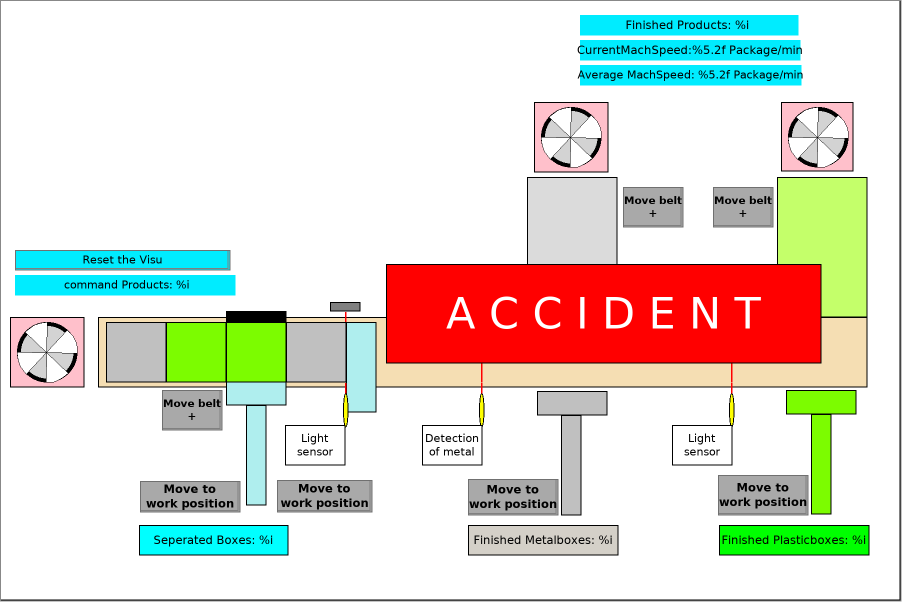
VISUALIZATION VIS_TemplateMachine  // 902x602
    Rectangle (0,0 900x600)
    Rectangle (98,317 769x70)
    Rectangle (777,177 90x140)
    Rectangle (527,177 90x140)
    Rectangle (716,302 30x9)
    Rectangle (467,302 30x9)
    Ellipse (479,393 5x34)
    Ellipse (729,393 5x34)
    Group (537,391 70x124)
        p2738717112: MAIN.fbVisu.fYMetal
        Rectangle (0,0 70x24)
        Rectangle (24,24 20x100)
    Group (787,391 70x124)
        p2738717112: MAIN.fbVisu.fYPlastic
        Rectangle (-1,-1 70x24)
        Rectangle (24,23 20x100)
    Group (227,382 60x124)
        p2738717112: MAIN.fbVisu.fYClamp
        Rectangle (19,23 20x100)
        Rectangle (-1,-1 60x24)
    Rectangle (106,322 60x60)
        p3560616238: MAIN.fbVisu.aBoxX[4]
        p2738717112: MAIN.fbVisu.aBoxY[4]
    Rectangle (226,322 60x60)
        p3560616238: MAIN.fbVisu.aBoxX[2]
        p2738717112: MAIN.fbVisu.aBoxY[2]
    Rectangle (166,322 60x60)
        p3560616238: MAIN.fbVisu.aBoxX[3]
        p2738717112: MAIN.fbVisu.aBoxY[3]
    Textfield (422,425 60x40), "Detection of metal"
    Textfield (672,425 60x40), "Light sensor"
    Rectangle (481,383 1x10)
    Rectangle (481,312 1x70)
    Rectangle (731,312 1x70)
    Rectangle (731,383 1x10)
    Button (623,187 60x40), "Move belt +", colour toggle: MAIN.fbVisu.bButtonColorMetalFw, invisible if: NOT (MAIN.fbMachine.eMode= 3), input disabled if: NOT (MAIN.fbMachine.eState = ePMLState_Execute)
        p573394764: MAIN.fbVisu.nButtonColorMetalFw
        toggle MAIN.fbVisu.bButtonMetalFwOut
    Button (713,187 60x40), "Move belt +", colour toggle: MAIN.fbVisu.bButtonColorPlasticFw, invisible if: NOT (MAIN.fbMachine.eMode= 3), input disabled if: NOT (MAIN.fbMachine.eState = ePMLState_Execute)
        p573394764: MAIN.fbVisu.nButtonColorPlasticFw
        toggle MAIN.fbVisu.bButtonPlasticFwOut
    Button (162,390 60x40), "Move belt +", colour toggle: MAIN.fbVisu.bButtonColorMainFw, invisible if: NOT (MAIN.fbMachine.eMode= 3), input disabled if: NOT (MAIN.fbMachine.eState = ePMLState_Execute)
        p573394764: MAIN.fbVisu.nButtonColorMainFw
        toggle MAIN.fbVisu.bButtonMainFwOut
    Button (277,480 95x32), "Move to work position", colour toggle: MAIN.fbVisu.bButtonColorBarrier, invisible if: NOT (MAIN.fbMachine.eMode= 3), input disabled if: NOT (MAIN.fbMachine.eState = ePMLState_Execute)
        p573394764: MAIN.fbVisu.nButtonColorBarrier
        toggle MAIN.fbVisu.bButtonBarrierToWorkOut
    Button (140,481 100x31), "Move to work position", colour toggle: MAIN.fbVisu.bButtonColorClamp, invisible if: NOT (MAIN.fbMachine.eMode= 3), input disabled if: NOT (MAIN.fbMachine.eState = ePMLState_Execute)
        p573394764: MAIN.fbVisu.nButtonColorClamp
        toggle MAIN.fbVisu.bButtonClampToWorkOut
    Button (468,479 90x36), "Move to work position", colour toggle: MAIN.fbVisu.bButtonColorMetalCyl, invisible if: NOT (MAIN.fbMachine.eMode= 3), input disabled if: NOT (MAIN.fbMachine.eState = ePMLState_Execute)
        p573394764: MAIN.fbVisu.nButtonColorMetalCyl
        toggle MAIN.fbVisu.bButtonMetalToWorkOut
    Button (718,475 90x40), "Move to work position", colour toggle: MAIN.fbVisu.bButtonColorPlasticCyl, invisible if: NOT (MAIN.fbMachine.eMode= 3), input disabled if: NOT (MAIN.fbMachine.eState = ePMLState_Execute)
        p573394764: MAIN.fbVisu.nButtonColorPlasticCyl
        toggle MAIN.fbVisu.bButtonPlasticToWorkOut
    Rectangle (346,322 30x90)
        p2738717112: MAIN.fbVisu.fYBarrier
    Rectangle (330,302 30x9)
    Ellipse (343,393 5x34)
    Rectangle (345,383 1x10)
    Rectangle (345,312 1x70)
    Textfield (285,425 60x40), "Light sensor"
    Rectangle (226,311 60x11)
    Rectangle (286,322 60x60)
        p3560616238: MAIN.fbVisu.aBoxX[1]
        p2738717112: MAIN.fbVisu.aBoxY[1]
    Rectangle (386,264 435x99), "A C C I D E N T", invisible if: NOT MAIN.fbVisu.bAccident
    Textfield (10,317 74x70)
    Rectangle (46,322 1x60)
    Rectangle (17,352 60x1)
    Ellipse (17,322 60x60)
    Polygon (47,322) (46,382) (53,382) (58,380) (63,377) (68,373) (25,332) (22,336) (20,340) (18,345) (17,352) (77,353) (77,347) (76,342) (73,336) (67,330) (26,374) (23,370) (20,366) (18,360) (17,353) (18,347) (19,342) (22,336) (26,331) (30,328) (34,325) (40,323)
        p2858320360: MAIN.fbVisu.nAngleMain
    Textfield (534,102 74x70)
    Rectangle (570,107 1x60)
    Rectangle (541,137 60x1)
    Ellipse (541,107 60x60)
    Polygon (571,107) (570,167) (577,167) (582,165) (587,162) (592,158) (549,117) (546,121) (544,125) (542,130) (541,137) (601,138) (601,132) (600,127) (597,121) (591,115) (550,159) (547,155) (544,151) (542,145) (541,138) (542,132) (543,127) (546,121) (550,116) (554,113) (558,110) (564,108)
        p2858320360: MAIN.fbVisu.nAngleMetal
    Textfield (781,102 72x69)
    Rectangle (817,107 1x60)
    Rectangle (788,137 60x1)
    Ellipse (788,107 60x60)
    Polygon (818,107) (817,167) (824,167) (829,165) (834,162) (839,158) (796,117) (793,121) (791,125) (789,130) (788,137) (848,138) (848,132) (847,127) (844,121) (838,115) (797,159) (794,155) (791,151) (789,145) (788,138) (789,132) (790,127) (793,121) (797,116) (801,113) (805,110) (811,108)
        p2858320360: MAIN.fbVisu.nAnglePlastic
    Rectangle (15,275 220x20), "command Products: %i", text variable: PackTags.Command.Parameter[2].Value, colour toggle: (MAIN.fbVisu.bInValidEntry OR PackTags.Admin.Warning[1].Trigger), invisible if: NOT ( MAIN.fbMachine.eMode = 1)
        OnMouseClick: write nVisuProductCommand via Default
    Rectangle (580,15 218x20), "Finished Products: %i", text variable: PackTags.Admin.ProdProcessedCount[1].Count, invisible if: NOT ( MAIN.fbMachine.eMode = 1)
    Button (15,250 215x20), "Reset the Visu", invisible if: (MAIN.fbMachine.eMode = 1 AND (MAIN.fbMachine.eState = ePMLState_Clearing OR MAIN.fbMachine.eState = ePMLState_Aborting OR MAIN.fbMachine.eState = ePMLState_Stopping OR MAIN.fbMachine.eState = ePMLState_Resetting OR MAIN.fbMachine.eState = ePMLState_Starting OR MAIN.fbMachine.eState = ePMLState_Execute OR MAIN.fbMachine.eState = ePMLState_Completing OR MAIN.fbMachine.eState = ePMLState_Suspending OR MAIN.fbMachine.eState = ePMLState_Holding))
        tap stChangeIntoProduction.bYesReset
    Rectangle (580,40 220x20), "CurrentMachSpeed:%5.2f Package/min", text variable: PackTags.Status.CurMachineSpeed, invisible if: NOT ( MAIN.fbMachine.eMode = 1)
    Rectangle (468,525 150x30), "Finished Metalboxes: %i", text variable: PackTags.Admin.ProdProcessedCount[4].Count, invisible if: NOT ( MAIN.fbMachine.eMode = 1)
    Rectangle (719,525 150x30), "Finished Plasticboxes: %i", text variable: PackTags.Admin.ProdProcessedCount[3].Count, invisible if: NOT ( MAIN.fbMachine.eMode = 1)
    Rectangle (580,65 221x20), "Average MachSpeed: %5.2f Package/min", text variable: PackTags.Status.MachineSpeed, invisible if: NOT ( MAIN.fbMachine.eMode = 1)
    Rectangle (139,525 149x30), "Seperated Boxes: %i", text variable: PackTags.Admin.ProdProcessedCount[2].Count, invisible if: NOT ( MAIN.fbMachine.eMode = 1)
END_VISUALIZATION

(* stored: Version 1.1.0.1
   Visu VIS_TemplateMachine: Id {9421e918-9a93-4f23-9733-2bf87c96933b} *)
